PROGRAM P_Circle
VAR
	iEndNumberCircle	:INT;(*書き終わった円の個数*)
	iWrittingCircle		:INT;(*今から何個目の円を書くのか*)
	i					:INT;
	stCircleSettings	:ARRAY[1..32] OF ST_CircleSettings;
	
	eStep				:E_CircleWriteStep:=E_CircleWriteStep.Check;
	iStep				:INT:=0;
	lrDeg				:LREAL :=0;

	fbMCMoveAbsolute0	:ARRAY[E_Axis.X_Axis..E_Axis.Z_Axis] OF MC_MoveAbsolute;
	fbMCMoveAbsolute1	:ARRAY[E_Axis.X_Axis..E_Axis.Z_Axis] OF MC_MoveAbsolute;
	MoveAbsoluteOut0	:ARRAY[E_Axis.X_Axis..E_Axis.Z_Axis] OF ST_McOutputs;
	MoveAbsoluteOut1	:ARRAY[E_Axis.X_Axis..E_Axis.Z_Axis] OF ST_McOutputs;
	fbZAxisTPCon0		:FB_Z_Axis_TargetPositionConvert;
	fbZAxisTPCon1		:FB_Z_Axis_TargetPositionConvert;
	bCheck0				:ARRAY[E_Axis.X_Axis..E_Axis.Z_Axis] OF BOOL;
	bCheck1				:ARRAY[E_Axis.X_Axis..E_Axis.Z_Axis] OF BOOL;
END_VAR

CASE eStep OF

E_CircleWriteStep.Check:(*まず書く円を確認*)

	iEndNumberCircle:=iWrittingCircle;
	iWrittingCircle:=0;

	FOR i :=  iEndNumberCircle + 1 TO 32 BY 1 DO
		IF stCircleSettings[i].bWrite=TRUE THEN
			iWrittingCircle:=i;
			eStep:=E_CircleWriteStep.First_Potision_Move;
			EXIT;
		END_IF
	END_FOR

	IF iWrittingCircle=0 THEN
		GVL_Motion.bCircleWriteFin:=TRUE;
	END_IF

E_CircleWriteStep.First_Potision_Move:(*円の書き始め位置へ移動*)

	CASE iStep OF
	0:
		iStep:=1;
		lrDeg:=stCircleSettings[iWrittingCircle].lrStartDeg;
		
	1:
		fbMCMoveAbsolute0[E_Axis.X_Axis].Execute:=TRUE;
		fbMCMoveAbsolute0[E_Axis.Y_Axis].Execute:=TRUE;
		fbMCMoveAbsolute0[E_Axis.X_Axis].Position:=stCircleSettings[iWrittingCircle].uiXCenter + stCircleSettings[iWrittingCircle].uiRadius * COS(lrDeg*PI/180);
		fbMCMoveAbsolute0[E_Axis.Y_Axis].Position:=stCircleSettings[iWrittingCircle].uiYCenter + stCircleSettings[iWrittingCircle].uiRadius * SIN(lrDeg*PI/180);
		fbMCMoveAbsolute0[E_Axis.X_Axis].Velocity:=150;
		fbMCMoveAbsolute0[E_Axis.Y_Axis].Velocity:=150;

		IF MoveAbsoluteOut0[E_Axis.X_Axis].Done=TRUE AND MoveAbsoluteOut0[E_Axis.Y_Axis].Done=TRUE THEN
			iStep:=2;
			fbMCMoveAbsolute0[E_Axis.X_Axis].Execute:=FALSE;
			fbMCMoveAbsolute0[E_Axis.Y_Axis].Execute:=FALSE;
		END_IF;
		
	2:
		fbMCMoveAbsolute0[E_Axis.Z_Axis].Execute:=TRUE;
		fbMCMoveAbsolute0[E_Axis.Z_Axis].Velocity:=150;
		
		fbZAxisTPCon0(
			lrX_AxisTP		:=fbMCMoveAbsolute0[E_Axis.X_Axis].Position,
			lrY_AxisTP		:=fbMCMoveAbsolute0[E_Axis.Y_Axis].Position,
			lrZ_AxisTP		:=273-GVL.lrPenFullLength+GVL.lrPenGripLength,
			lrZ_AxisCorTP	=>fbMCMoveAbsolute0[E_Axis.Z_Axis].Position
			);
				
		IF MoveAbsoluteOut0[E_Axis.Z_Axis].Done=TRUE THEN
			eStep:=E_CircleWriteStep.Write_Circle;
			fbMCMoveAbsolute0[E_Axis.Z_Axis].Execute:=FALSE;
			iStep:=0;
		END_IF;
	
	END_CASE;

E_CircleWriteStep.Write_Circle:(*円を書いていく*)

	CASE iStep OF
	0:
		bCheck0[E_Axis.X_Axis]:=TRUE;
		bCheck1[E_Axis.X_Axis]:=TRUE;
		bCheck0[E_Axis.Y_Axis]:=TRUE;
		bCheck1[E_Axis.Y_Axis]:=TRUE;
		bCheck0[E_Axis.Z_Axis]:=TRUE;
		bCheck1[E_Axis.Z_Axis]:=TRUE;
		lrDeg:=stCircleSettings[iWrittingCircle].lrStartDeg;
		iStep:=1;

	1:	
		IF MoveAbsoluteOut0[E_Axis.X_Axis].Done=TRUE THEN bCheck0[E_Axis.X_Axis]:=TRUE; END_IF;
		IF MoveAbsoluteOut1[E_Axis.X_Axis].Done=TRUE THEN bCheck1[E_Axis.X_Axis]:=TRUE; END_IF;
		IF MoveAbsoluteOut0[E_Axis.Y_Axis].Done=TRUE THEN bCheck0[E_Axis.Y_Axis]:=TRUE; END_IF;
		IF MoveAbsoluteOut1[E_Axis.Y_Axis].Done=TRUE THEN bCheck1[E_Axis.Y_Axis]:=TRUE; END_IF;
		IF MoveAbsoluteOut0[E_Axis.Z_Axis].Done=TRUE THEN bCheck0[E_Axis.Z_Axis]:=TRUE; END_IF;
		IF MoveAbsoluteOut1[E_Axis.Z_Axis].Done=TRUE THEN bCheck1[E_Axis.Z_Axis]:=TRUE; END_IF;
	
		IF bCheck0[E_Axis.X_Axis]=TRUE AND bCheck0[E_Axis.Y_Axis]=TRUE AND bCheck0[E_Axis.Z_Axis]=TRUE THEN
			bCheck0[E_Axis.X_Axis]:=FALSE;	
			bCheck0[E_Axis.Y_Axis]:=FALSE;
			bCheck0[E_Axis.Z_Axis]:=FALSE;
			lrDeg:=lrDeg + 1;
			fbMCMoveAbsolute0[E_Axis.X_Axis].Position:=stCircleSettings[iWrittingCircle].uiXCenter + stCircleSettings[iWrittingCircle].uiRadius * COS(lrDeg*PI/180);
			fbMCMoveAbsolute0[E_Axis.Y_Axis].Position:=stCircleSettings[iWrittingCircle].uiYCenter + stCircleSettings[iWrittingCircle].uiRadius * SIN(lrDeg*PI/180);
			
			fbZAxisTPCon0(
				lrX_AxisTP		:=fbMCMoveAbsolute0[E_Axis.X_Axis].Position,
				lrY_AxisTP		:=fbMCMoveAbsolute0[E_Axis.Y_Axis].Position,
				lrZ_AxisTP		:=273-GVL.lrPenFullLength+GVL.lrPenGripLength,
				lrZ_AxisCorTP	=>fbMCMoveAbsolute0[E_Axis.Z_Axis].Position
				);

			fbMCMoveAbsolute0[E_Axis.X_Axis].Execute:=TRUE;
			fbMCMoveAbsolute0[E_Axis.Y_Axis].Execute:=TRUE;
			fbMCMoveAbsolute0[E_Axis.Z_Axis].Execute:=TRUE;
			fbMCMoveAbsolute0[E_Axis.X_Axis].Velocity:=150;
			fbMCMoveAbsolute0[E_Axis.Y_Axis].Velocity:=150;
			fbMCMoveAbsolute0[E_Axis.Z_Axis].Velocity:=150;
		ELSE
			fbMCMoveAbsolute0[E_Axis.X_Axis].Execute:=FALSE;
			fbMCMoveAbsolute0[E_Axis.Y_Axis].Execute:=FALSE;
			fbMCMoveAbsolute0[E_Axis.Z_Axis].Execute:=FALSE;
		END_IF;
		
		IF bCheck1[E_Axis.X_Axis]=TRUE AND bCheck1[E_Axis.Y_Axis]=TRUE AND bCheck1[E_Axis.Z_Axis]=TRUE THEN
			bCheck1[E_Axis.X_Axis]:=FALSE;	
			bCheck1[E_Axis.Y_Axis]:=FALSE;
			bCheck1[E_Axis.Z_Axis]:=FALSE;
			lrDeg:=lrDeg + 1;
			fbMCMoveAbsolute1[E_Axis.X_Axis].Position:=stCircleSettings[iWrittingCircle].uiXCenter + stCircleSettings[iWrittingCircle].uiRadius * COS(lrDeg*PI/180);
			fbMCMoveAbsolute1[E_Axis.Y_Axis].Position:=stCircleSettings[iWrittingCircle].uiYCenter + stCircleSettings[iWrittingCircle].uiRadius * SIN(lrDeg*PI/180);
			
			fbZAxisTPCon1(
				lrX_AxisTP		:=fbMCMoveAbsolute1[E_Axis.X_Axis].Position,
				lrY_AxisTP		:=fbMCMoveAbsolute1[E_Axis.Y_Axis].Position,
				lrZ_AxisTP		:=273-GVL.lrPenFullLength+GVL.lrPenGripLength,
				lrZ_AxisCorTP	=>fbMCMoveAbsolute1[E_Axis.Z_Axis].Position
				);

			fbMCMoveAbsolute1[E_Axis.X_Axis].Execute:=TRUE;
			fbMCMoveAbsolute1[E_Axis.Y_Axis].Execute:=TRUE;
			fbMCMoveAbsolute1[E_Axis.Z_Axis].Execute:=TRUE;
			fbMCMoveAbsolute1[E_Axis.X_Axis].Velocity:=150;
			fbMCMoveAbsolute1[E_Axis.Y_Axis].Velocity:=150;
			fbMCMoveAbsolute1[E_Axis.Z_Axis].Velocity:=150;
		ELSE
			fbMCMoveAbsolute1[E_Axis.X_Axis].Execute:=FALSE;
			fbMCMoveAbsolute1[E_Axis.Y_Axis].Execute:=FALSE;
			fbMCMoveAbsolute1[E_Axis.Z_Axis].Execute:=FALSE;
		END_IF;
	
		IF stCircleSettings[iWrittingCircle].lrEndDeg < lrDeg THEN
			fbMCMoveAbsolute0[E_Axis.X_Axis].Execute:=FALSE;
			fbMCMoveAbsolute0[E_Axis.Y_Axis].Execute:=FALSE;
			fbMCMoveAbsolute0[E_Axis.Z_Axis].Execute:=FALSE;
			fbMCMoveAbsolute1[E_Axis.X_Axis].Execute:=FALSE;
			fbMCMoveAbsolute1[E_Axis.Y_Axis].Execute:=FALSE;
			fbMCMoveAbsolute1[E_Axis.Z_Axis].Execute:=FALSE;
			eStep:=E_CircleWriteStep.Z_Axix_Up_Potision;
			iStep:=0;
			lrDeg:=0;
		END_IF;
	
	END_CASE;

E_CircleWriteStep.Z_Axix_Up_Potision:(*Z軸を持ち上げる、ペンが紙に当たらないように*)

	fbMCMoveAbsolute0[E_Axis.Z_Axis].Execute:=TRUE;
	fbMCMoveAbsolute0[E_Axis.Z_Axis].Position:=273-GVL.lrPenFullLength+GVL.lrPenGripLength-50;
	fbMCMoveAbsolute0[E_Axis.Z_Axis].Velocity:=150;

	IF MoveAbsoluteOut0[E_Axis.Z_Axis].Done=TRUE THEN
		eStep:=E_CircleWriteStep.Check;
		fbMCMoveAbsolute0[E_Axis.Z_Axis].Execute:=FALSE;
	END_IF;

END_CASE;

aMotion();

ACTION aMotion:
	fbMCMoveAbsolute0[E_Axis.X_Axis](
		Axis			:=GVL_Axis.stAxis[E_Axis.X_Axis],
		Execute			:=fbMCMoveAbsolute0[E_Axis.X_Axis].Execute,
		Position		:=fbMCMoveAbsolute0[E_Axis.X_Axis].Position,
		Velocity		:=fbMCMoveAbsolute0[E_Axis.X_Axis].Velocity,
		BufferMode		:=MC_BlendingNext,
		Done			=>MoveAbsoluteOut0[E_Axis.X_Axis].Done,
		Busy			=>MoveAbsoluteOut0[E_Axis.X_Axis].Busy,
		Active			=>MoveAbsoluteOut0[E_Axis.X_Axis].Active,
		CommandAborted	=>MoveAbsoluteOut0[E_Axis.X_Axis].CommandAborted,
		Error			=>MoveAbsoluteOut0[E_Axis.X_Axis].Error,
		ErrorID			=>MoveAbsoluteOut0[E_Axis.X_Axis].ErrorID
	);
		
	fbMCMoveAbsolute1[E_Axis.X_Axis](
		Axis			:=GVL_Axis.stAxis[E_Axis.X_Axis],
		Execute			:=fbMCMoveAbsolute1[E_Axis.X_Axis].Execute,
		Position		:=fbMCMoveAbsolute1[E_Axis.X_Axis].Position,
		Velocity		:=fbMCMoveAbsolute1[E_Axis.X_Axis].Velocity,
		BufferMode		:=MC_BlendingNext,
		Done			=>MoveAbsoluteOut1[E_Axis.X_Axis].Done,
		Busy			=>MoveAbsoluteOut1[E_Axis.X_Axis].Busy,
		Active			=>MoveAbsoluteOut1[E_Axis.X_Axis].Active,
		CommandAborted	=>MoveAbsoluteOut1[E_Axis.X_Axis].CommandAborted,
		Error			=>MoveAbsoluteOut1[E_Axis.X_Axis].Error,
		ErrorID			=>MoveAbsoluteOut1[E_Axis.X_Axis].ErrorID
	);

	fbMCMoveAbsolute0[E_Axis.Y_Axis](
		Axis			:=GVL_Axis.stAxis[E_Axis.Y_Axis],
		Execute			:=fbMCMoveAbsolute0[E_Axis.Y_Axis].Execute,
		Position		:=fbMCMoveAbsolute0[E_Axis.Y_Axis].Position,
		Velocity		:=fbMCMoveAbsolute0[E_Axis.Y_Axis].Velocity,
		BufferMode		:=MC_BlendingNext,
		Done			=>MoveAbsoluteOut0[E_Axis.Y_Axis].Done,
		Busy			=>MoveAbsoluteOut0[E_Axis.Y_Axis].Busy,
		Active			=>MoveAbsoluteOut0[E_Axis.Y_Axis].Active,
		CommandAborted	=>MoveAbsoluteOut0[E_Axis.Y_Axis].CommandAborted,
		Error			=>MoveAbsoluteOut0[E_Axis.Y_Axis].Error,
		ErrorID			=>MoveAbsoluteOut0[E_Axis.Y_Axis].ErrorID
	);

	fbMCMoveAbsolute1[E_Axis.Y_Axis](
		Axis			:=GVL_Axis.stAxis[E_Axis.Y_Axis],
		Execute			:=fbMCMoveAbsolute1[E_Axis.Y_Axis].Execute,
		Position		:=fbMCMoveAbsolute1[E_Axis.Y_Axis].Position,
		Velocity		:=fbMCMoveAbsolute1[E_Axis.Y_Axis].Velocity,
		BufferMode		:=MC_BlendingNext,
		Done			=>MoveAbsoluteOut1[E_Axis.Y_Axis].Done,
		Busy			=>MoveAbsoluteOut1[E_Axis.Y_Axis].Busy,
		Active			=>MoveAbsoluteOut1[E_Axis.Y_Axis].Active,
		CommandAborted	=>MoveAbsoluteOut1[E_Axis.Y_Axis].CommandAborted,
		Error			=>MoveAbsoluteOut1[E_Axis.Y_Axis].Error,
		ErrorID			=>MoveAbsoluteOut1[E_Axis.Y_Axis].ErrorID
	);

	fbMCMoveAbsolute0[E_Axis.Z_Axis](
		Axis			:=GVL_Axis.stAxis[E_Axis.Z_Axis],
		Execute			:=fbMCMoveAbsolute0[E_Axis.Z_Axis].Execute,
		Position		:=fbMCMoveAbsolute0[E_Axis.Z_Axis].Position,
		Velocity		:=fbMCMoveAbsolute0[E_Axis.Z_Axis].Velocity,
		BufferMode		:=MC_BlendingNext,
		Done			=>MoveAbsoluteOut0[E_Axis.Z_Axis].Done,
		Busy			=>MoveAbsoluteOut0[E_Axis.Z_Axis].Busy,
		Active			=>MoveAbsoluteOut0[E_Axis.Z_Axis].Active,
		CommandAborted	=>MoveAbsoluteOut0[E_Axis.Z_Axis].CommandAborted,
		Error			=>MoveAbsoluteOut0[E_Axis.Z_Axis].Error,
		ErrorID			=>MoveAbsoluteOut0[E_Axis.Z_Axis].ErrorID
	);
	
	fbMCMoveAbsolute1[E_Axis.Z_Axis](
		Axis			:=GVL_Axis.stAxis[E_Axis.Z_Axis],
		Execute			:=fbMCMoveAbsolute1[E_Axis.Z_Axis].Execute,
		Position		:=fbMCMoveAbsolute1[E_Axis.Z_Axis].Position,
		Velocity		:=fbMCMoveAbsolute1[E_Axis.Z_Axis].Velocity,
		BufferMode		:=MC_BlendingNext,
		Done			=>MoveAbsoluteOut1[E_Axis.Z_Axis].Done,
		Busy			=>MoveAbsoluteOut1[E_Axis.Z_Axis].Busy,
		Active			=>MoveAbsoluteOut1[E_Axis.Z_Axis].Active,
		CommandAborted	=>MoveAbsoluteOut1[E_Axis.Z_Axis].CommandAborted,
		Error			=>MoveAbsoluteOut1[E_Axis.Z_Axis].Error,
		ErrorID			=>MoveAbsoluteOut1[E_Axis.Z_Axis].ErrorID
	);
END_ACTION

END_PROGRAM

(* stored: Version 1.1.0.1, ProductVersion 3.1.4024.12
   POU P_Circle: Id {8197147f-2da7-42d5-b34c-a65de439fcff}, SpecialFunc None
   Action aMotion: Id {c6a78444-7f7e-404b-b879-43f4ce9a1ec7} *)
